FUNCTION_BLOCK "fbArchiveEquipRectifier"
{ S7_Optimized_Access := 'TRUE' }
VERSION : 0.8
   VAR
      equipmentRectifier { ExternalWritable := 'False'} : Array[1..1] of "tEquipment";
   END_VAR

   VAR_TEMP
      tempInt : Int;
   END_VAR


BEGIN
END_FUNCTION_BLOCK

